Universal Robots PolyScope program: mqtt-ur3-bridge-main.urp

Program mqtt-ur3-bridge-main (installation=mqtt-ur3-bridge-installation directory=/programs/mqtt-ur3-bridge createdIn=5.12.4.1101661 lastSavedIn=5.12.4.1101661 robotSerialNumber=20225390026)
Calibrated DH parameters: a=[-0.00006, -0.174938, -0.210866, 0.000084, -0.000074, 0]; d=[0.152034, 47.601021, -53.624686, 6.154381, 0.08549, 0.092322]; alpha=[1.570162, -0.003579, 0.005473, 1.573232, -1.570689, 0]; deltaTheta=[0, -0.772192, 0.617109, 0.155089, 0.000002, 0]
BeforeStart
  val := "nA"
  cmd := "nA"
  smoothGain := 200
  smoothRate := 0.1
  isInterpretm := False
  isRpiSocketOpen := False
  isRpiOn := False
  isFree := False
  isFreeLast := True
  SuppressedNode
    MoveJ speed 60 deg/s, acceleration 80 deg/s^2 (useActiveTCP=true) feature=Base
      'reative movement of 0mm to circumvent ISO norm.'
      Waypoint relative_start (Relative): relativeFromPosition TCP in base x=12.337 y=-373.169 z=695.383 mm, rx=3.1376 ry=0.0316 rz=0.0129 rad; joints [2.032, -90.023, 0.001, -89.999, 0.003, 0] deg; TCP offset x=0 y=0 z=150 mm, rx=-0.0044 ry=-2.2082 rz=-2.2136 rad; TCP in base x=-1.299 y=-373.374 z=695.381 mm, rx=3.1375 ry=-0.0224 rz=0.0151 rad; joints [0.061, -89.94, 0, -89.998, 0.001, -0.001] deg
  MoveJ speed 60 deg/s, acceleration 80 deg/s^2 (useActiveTCP=true) feature=Base
    'absolute hom'
    Waypoint home: TCP in base x=132.575 y=379.691 z=475.417 mm, rx=0.0122 ry=3.1147 rz=-0.0253 rad; joints [89, -89.381, -91.565, -0.14, 91.052, 718.308] deg; TCP offset x=0 y=0 z=77 mm, rx=-0.0044 ry=-2.2082 rz=-2.2136 rad
Robot Program (runOnlyOnce=false)
  Loop While (checkContinuously=false) expression=isInterpretm≟ False
    'normal operation'
    Loop While (checkContinuously=false) expression=isNewMjJoints
      isNewMjJoints := False
      If val≟"nA"
        Script: movej(targetJoints,acc,vel,0,0)
      If val≟"blend"
        Script: movej(targetJoints,acc,vel,0,blend)
      If val≟"time"
        Script: movej(targetJoints,1,1,time,0)
      If val≟"time,blend" or val≟"blend,time"
        Script: movej(targetJoints,1,1,time,blend)
    Loop While (checkContinuously=false) expression=isNewMjPose
      isNewMjPose := False
      If get_inverse_kin_has_solution(targetPose)
        If val≟"nA"
          Script: movej(targetPose,acc,vel,0,0)
        If val≟"blend"
          Script: movej(targetPose,acc,vel,0,blend)
        If val≟"time"
          Script: movej(targetPose,1,1,time,0)
        If val≟"time,blend" or val≟"blend,time"
          Script: movej(targetPose,1,1,time,blend)
      Else 
        Script: socket_send_line("return:can't reach the requested pose. Do nthng","rpi")
        MoveJ speed 60 deg/s, acceleration 80 deg/s^2 (useActiveTCP=true) feature=Base
          Waypoint shortup (Relative): motionParameters(jointSpeed=1.745329 jointAcceleration=17.453293 cartesianSpeed=0.25 cartesianAcceleration=1.2); relativeFromPosition TCP in base x=248.981 y=-243.921 z=117.024 mm, rx=-3.1056 ry=0.3562 rz=-0.0688 rad; joints [-23.13, -103.26, -108.87, -55.69, -268.376, 260.446] deg; TCP offset x=-4.416 y=0.714 z=70.405 mm, rx=0 ry=0 rz=0 rad; TCP in base x=259.787 y=-248.579 z=130.586 mm, rx=-3.1141 ry=0.3568 rz=-0.1226 rad; joints [-23.132, -103.279, -105.63, -56.867, -268.375, 260.444] deg
          Waypoint shortdown (Relative): motionParameters(jointSpeed=1.745329 jointAcceleration=17.453293 cartesianSpeed=0.25 cartesianAcceleration=1.2); relativeFromPosition TCP in base x=259.786 y=-248.578 z=130.588 mm, rx=-3.1141 ry=0.3568 rz=-0.1226 rad; joints [-23.132, -103.278, -105.629, -56.868, -268.375, 260.447] deg; TCP in base x=248.978 y=-243.921 z=117.009 mm, rx=-3.1056 ry=0.3562 rz=-0.0687 rad; joints [-23.13, -103.263, -108.87, -55.69, -268.376, 260.445] deg
    Loop While (checkContinuously=false) expression=isNewSpeedl
      isNewSpeedl := False
      Script: speedl(newSpeedl,1.0,0.2)
    Loop While (checkContinuously=false) expression=isNewSmoothPose
      isNewSmoothPose := False
      Script: servoj(get_inverse_kin(newSmoothPose),0,0,smoothRate,smoothGain)
    Loop While (checkContinuously=false) expression=isNewSmoothJoi
      isNewSmoothJoi := False
      Script: servoj(newSmoothJoints,0,0,smoothRate,smoothGain)
    If isFree≠isFreeLast
      If isFree
        Script: freedrive_mode()
      Else 
        Script: end_freedrive_mode()
      isFreeLast := isFree
    'if nthng happens, wait to cool down main'
    Wait Sleep waitTime=0.01
  Loop While (checkContinuously=true) expression=isInterpretm
    Wait Sleep waitTime=0.1
    isInterpretm := False
    Script: interpreter_mode()
  'if nthng happens, wait to cool down main'
  Wait Sleep waitTime=0.01
Thread Thread_1 (runOnlyOnce=false)
  'THREAD for socket coonection to RPI'
  Timer (action=Start) variable(name=timer_socket)
  Timer (action=Start) variable(name=timer_lastRpiOn)
  Loop Forever
    If isRpiSocketOpen≟ False
      Script: socket_close(socket_name="rpi")
      Wait Sleep waitTime=0.5
      isRpiSocketOpen := socket_open("10.3.3.1",30001,"rpi")
      If isRpiSocketOpen≟ True
        Timer (action=Reset) variable=timer_socket
        Script: socket_send_string("ur3Online","rpi")
      Else 
        Wait Sleep waitTime=2
    Else 
      'IF Rpi Socket is open:'
      If timer_socket>2
        'send status msg to rpi evey 2s'
        Script: socket_send_string("ur3Online","rpi")
        Timer (action=Reset) variable=timer_socket
      incoming_buff := socket_read_line("rpi")
      If incoming_buff≠""
        If incoming_buff≟"rpiOnline"
          isRpiOn := True
          Timer (action=Reset) variable=timer_lastRpiOn
        ElseIf incoming_buff≟"getStatus"
          Script: socket_send_string("gotStatus","rpi")
        Else 
          colPos := str_find(incoming_buff,":")
          Script: socket_send_line(str_cat("ur3executes:",incoming_buff),"rpi")
          If colPos≥0
            cmd := str_sub(incoming_buff,0,colPos)
            val := str_sub(incoming_buff,colPos+1,str_len(incoming_buff))
            If val≟""
              val := "nA"
            If cmd≟"pause"
              stop_mov := True
            If cmd≟"continue"
              stop_mov := False
          If colPos≟-1
            cmd := incoming_buff
            val := "nA"
      If timer_lastRpiOn>10
        isRpiOn := False
        isRpiSocketOpen := False
        Script: socket_close(socket_name="rpi")
    Wait Sleep waitTime=0.01
    Script: sync()
Thread Thread_2 (runOnlyOnce=false)
  'THREAD for internal socket coonection (speed)'
  isSpeedSockOpen := False
  Script: isSpeedSockOpen=socket_open("127.0.0.1",30002,"sps")
  Loop Forever
    If stop_mov≠stop_mov_last
      stop_mov := stop_mov*-1
      speed := "1"
      If stop_mov≟ True
        speed := "0.1"
      Script: socket_send_string("set speed","sps")
      Script: socket_send_string(speed,"sps")
      Script: socket_send_byte(10,"sps")
      stop_mov_last := stop_mov
    Wait Sleep waitTime=0.05
    Script: sync()
Thread Thread_3 (runOnlyOnce=false)
  'setting cmds'
  Loop Forever
    arrayPos := 0
    colArrayPos := 0
    If cmd≠"" or cmd≠"nA"
      If cmd≟"getPose"
        Script: actualPose=get_actual_tcp_pose()
        Script: socket_send_line(str_cat("returnValues:pose:",to_str(actualPose)),"rpi")
      ElseIf cmd≟"getJoints"
        Script: actualJoints=get_actual_joint_positions()
        Script: socket_send_line(str_cat("returnValues:joints:",to_str(actualJoints)),"rpi")
      ElseIf cmd≟"getForce"
        actualForce := get_tcp_force()
        Script: socket_send_line(str_cat("returnValues:force:",to_str(actualForce)),"rpi")
      ElseIf cmd≟"free" and val≟"start"
        isFree := True
      ElseIf cmd≟"free" and val≟"stop"
        isFree := False
      If cmd≟"joints" or cmd≟"jointsm"
        arrayVal := val
        Loop While (checkContinuously=false) expression=colArrayPos≥0
          colArrayPos := str_find(arrayVal,",")
          If colArrayPos<0
            Script: targetJoints[arrayPos]=to_num(arrayVal)
          Else 
            Script: targetJoints[arrayPos]=to_num(str_sub(arrayVal,0,colArrayPos))
            arrayVal := str_sub(arrayVal,colArrayPos+1,str_len(arrayVal))
          Script: arrayPos=arrayPos+1
        If cmd≟"jointsm"
          isNewMjPose := True
      ElseIf cmd≟"pose" or cmd≟"posem"
        arrayVal := val
        Loop While (checkContinuously=false) expression=colArrayPos≥0
          colArrayPos := str_find(arrayVal,",")
          If colArrayPos<0
            Script: targetPose[arrayPos]=to_num(arrayVal)
          Else 
            Script: targetPose[arrayPos]=to_num(str_sub(arrayVal,0,colArrayPos))
            arrayVal := str_sub(arrayVal,colArrayPos+1,str_len(arrayVal))
          Script: arrayPos=arrayPos+1
        If cmd≟"posem"
          isNewMjPose := True
      ElseIf cmd≟"contSpeed"
        arrayVal := val
        Loop While (checkContinuously=false) expression=colArrayPos≥0
          colArrayPos := str_find(arrayVal,",")
          If colArrayPos<0
            Script: newSpeedl[arrayPos]=to_num(arrayVal)
          Else 
            Script: newSpeedl[arrayPos]=to_num(str_sub(arrayVal,0,colArrayPos))
            arrayVal := str_sub(arrayVal,colArrayPos+1,str_len(arrayVal))
          Script: arrayPos=arrayPos+1
        isNewSpeedl := True
      ElseIf cmd≟"smoothPose"
        arrayVal := val
        Loop While (checkContinuously=false) expression=colArrayPos≥0
          colArrayPos := str_find(arrayVal,",")
          If colArrayPos<0
            Script: newSmoothPose[arrayPos]=to_num(arrayVal)
          Else 
            Script: newSmoothPose[arrayPos]=to_num(str_sub(arrayVal,0,colArrayPos))
            arrayVal := str_sub(arrayVal,colArrayPos+1,str_len(arrayVal))
          Script: arrayPos=arrayPos+1
        isNewSmoothPose := True
      ElseIf cmd≟"smoothJoints"
        arrayVal := val
        Loop While (checkContinuously=false) expression=colArrayPos≥0
          colArrayPos := str_find(arrayVal,",")
          If colArrayPos<0
            Script: newSmoothJoints[arrayPos]=to_num(arrayVal)
          Else 
            Script: newSmoothJoints[arrayPos]=to_num(str_sub(arrayVal,0,colArrayPos))
            arrayVal := str_sub(arrayVal,colArrayPos+1,str_len(arrayVal))
          Script: arrayPos=arrayPos+1
        isNewSmoothJoi := True
      ElseIf cmd≟"x"
        Script: targetPose[0]=to_num(val)
      ElseIf cmd≟"y"
        Script: targetPose[1]=to_num(val)
      ElseIf cmd≟"z"
        Script: targetPose[2]=to_num(val)
      ElseIf cmd≟"ax"
        Script: targetPose[3]=to_num(val)
      ElseIf cmd≟"ay"
        Script: targetPose[4]=to_num(val)
      ElseIf cmd≟"az"
        Script: targetPose[5]=to_num(val)
      ElseIf cmd≟"j1"
        Script: targetJoints[0]=to_num(val)
      ElseIf cmd≟"j2"
        Script: targetJoints[1]=to_num(val)
      ElseIf cmd≟"j3"
        Script: targetJoints[2]=to_num(val)
      ElseIf cmd≟"j4"
        Script: targetJoints[3]=to_num(val)
      ElseIf cmd≟"j5"
        Script: targetJoints[4]=to_num(val)
      ElseIf cmd≟"j6"
        Script: targetJoints[5]=to_num(val)
      ElseIf cmd≟"vel"
        Script: vel=to_num(val)
      ElseIf cmd≟"acc"
        Script: acc=to_num(val)
      ElseIf cmd≟"time"
        Script: time=to_num(val)
      ElseIf cmd≟"blend"
        Script: blend=to_num(val)
      ElseIf cmd≟"danceR"
        Script: danceR=to_num(val)
      ElseIf cmd≟"smoothGain"
        Script: smoothGain=to_num(val)
      ElseIf cmd≟"smoothRate"
        Script: smoothRate=to_num(val)
      ElseIf cmd≟"interpret"
        isInterpretm := True
      ElseIf cmd≟"movejPose"
        isNewMjPose := True
      ElseIf cmd≟"movejJoints"
        isNewMjJoints := True
      Else 
        Script: socket_send_string("cmdNotFound","rpi")
      cmd := "nA"
    SuppressedNode
      Wait Sleep waitTime=0.01
    Script: sync()
SuppressedNode
  Thread Thread_4 (runOnlyOnce=false)
    'Things that should happen while main thread is blocking'
    SuppressedNode
      Loop Forever
        If cmd≠"" or cmd≠"nA"
          Placeholder
        Wait Sleep waitTime=0.01
        Script: sync()
